FUNCTION_BLOCK SM_SafetyIO
VAR_INPUT
END_VAR
VAR_OUTPUT
	///Current status description
	{attribute 'OPC.UA.DA' := '1'}
	{attribute 'OPC.UA.DA.Access' := '1'}
	actualStatus: STRING;
	///Statuses of the state machine
	statuses: SafetyIOStatuses;
	///Parts of the state machine
	parts: SafetyIOParts;
END_VAR
VAR_IN_OUT
END_VAR
VAR
END_VAR

parts.domeAccess();
parts.hydraulicsAndSafety();
statuses.healthStatus(
    isGood := parts.hydraulicsAndSafety.statuses.healthStatus.isGood AND parts.domeAccess.statuses.healthStatus.isGood,
    hasWarning := parts.hydraulicsAndSafety.statuses.healthStatus.hasWarning OR parts.domeAccess.statuses.healthStatus.hasWarning);

END_FUNCTION_BLOCK

(* stored: Version 1.1.0.1, ProductVersion 3.1.4019.2
   POU SM_SafetyIO: Id {50cb1404-dfc5-41dc-89f4-dd372eae8140}, SpecialFunc None *)
